Fanuc KAREL source: kb00063.KL

PROGRAM KB00063
%STACKSIZE=65535
%PRIORITY=65535
%NOLOCKGROUP
VAR
P1 : INTEGER
P2 : INTEGER
P3 : INTEGER
BEGIN
P1=1
P2=1
P3=1
DEL_INST_TPE(P1,P2,P3)
END KB00063
